{attribute 'qualified_only'}
VAR_GLOBAL
END_VAR
VAR_GLOBAL
	// Pressure within the pumps
	nPressure: REAL := 1;
	// Whether the pump is on
	bPump: BOOL := FALSE;
END_VAR

(* stored: Version 1.1.0.1, ProductVersion 3.1.4024.12
   GVL GVL_Var: Id {86340a5d-f727-45f2-b9dd-2cf31392677f} *)
